{attribute 'GeneratedUsingTerminal: EP7402-0057-0017'}
{attribute addProperty BoxType "EP7402-0057-0017"}
{attribute addProperty Id "StatusAT %I*Status_725F98F27"}
{attribute addProperty CRC "2580668410"}
{attribute addProperty Size "7"}
TYPE STM_Status_Channel_99D1DFFA :
STRUCT
	{attribute addProperty Name "Status"}
	Status AT %I* : Status_725F98F2;
END_STRUCT
END_TYPE

(* stored: Version 1.2.0.0, ProductVersion 3.1.4024.9
   DUT STM_Status_Channel_99D1DFFA: Id {5282fd60-067d-4bf1-81c7-6f82a3a1dc66} *)
